{attribute 'pack_mode' := '2'}
TYPE ST_GEAR_DATA :
STRUCT
  rDeltaToMasterPos       : LREAL;
  rModuloSyncPosSlave     : LREAL;
  rMasterStartDistance    : LREAL;
  rGearNumerator          : LREAL;
  iGearDenumerator        : USINT  := 1;
END_STRUCT
END_TYPE

(* stored: Version 1.1.0.1
   DUT ST_GEAR_DATA: Id {d8fea0d2-788c-49cc-b90d-3264f31a8250} *)
